Fanuc KAREL source: ko00141.KL

-- PROVISIONAL review KL for V940-1; original PC SHA256 3835253479d16d6876b322fbb51adb467e7ca5bfb65cb2c12307dfc87141ccd1
-- Incomplete behavior may be omitted. Consult companion uncertainty JSON. Do not deploy.
PROGRAM KO00141
%NOLOCKGROUP
VAR
  R : REAL
  N : INTEGER
-- UNRESOLVED_DECL CFG type=00001c
-- UNRESOLVED_DECL OUT type=000102
BEGIN
  -- V9_ZERO_TABLE_METADATA_HINT layout=0001; no indexed target words; source/name/runtime held
  -- UNRESOLVED_PC offsets 5-12; opcodes 9D,23
  -- UNRESOLVED_PC offsets 17-28; opcodes 2E,23
  -- UNRESOLVED_PC offsets 33-43; opcodes 9D,22,A5
  -- UNRESOLVED_PC offsets 48-107; opcodes 27,22,22,22,27,21,64,22,22,22,76,7E,4A
  -- UNRESOLVED_PC offsets 112-116; opcodes 7F
END KO00141
